INTERFACE I_ComponentCollection EXTENDS I_Base

METHOD Accept
VAR_INPUT
	Visitor : I_ComponentVisitor;
END_VAR
END_METHOD

{attribute 'monitoring' := 'call'}
PROPERTY Count : UDINT
GET
END_GET
END_PROPERTY

METHOD GetAtIndex : I_Component
VAR_INPUT
	Index : UDINT;
END_VAR
END_METHOD

METHOD GetComponentByName : I_Component
VAR_INPUT
	Name : T_MaxString;
END_VAR
END_METHOD

END_INTERFACE

(* stored: Version 1.1.0.1, ProductVersion 3.1.4026.19
   Itf I_ComponentCollection: Id {cadf997f-6bee-48d5-b8f4-0a4cf5e22c66}
   Method Accept: Id {beafdad1-ed76-4206-a17e-6ca7f63f3670}
   Property Count: Id {cdbbc379-6b01-4e27-b9cf-c5d3cead7de7}
   Get Get: Id {5d87c04f-2e24-4afd-a569-d35860f1e484}
   Method GetAtIndex: Id {f7b9b9f2-6550-4554-b667-33eb61a3b7c1}
   Method GetComponentByName: Id {1f2dcbc9-b0c5-44ba-af82-138fa6441cc0} *)
